PROGRAM MAIN
VAR
	WeatherData : stWeatherData;
	bGetWeatherData : BOOL;
	sysTime : TIMESTRUCT;
	actDateTime : DT;
	fb_LocalSystemTime : FB_LocalSystemTime;
END_VAR

fb_LocalSystemTime(bEnable := TRUE, systemTime => sysTime);
actDateTime := SYSTEMTIME_TO_DT(sysTime);

IF actDateTime > WeatherData.Forecast[0].timeTo THEN
	bGetWeatherData := TRUE;
END_IF

END_PROGRAM

(* stored: Version 1.1.0.1, ProductVersion 3.1.4024.2
   POU MAIN: Id {555858ef-0c6a-4966-a768-92a29ef617b6}, SpecialFunc None *)
